RESOURCE_TYPE DM_RES (* Device Management Resource Type *)
  (* Standard: 61499-2 *)
  (* Version 0.0, 2000-05-27, JHC, Rockwell Automation *)
  VAR_INPUT
    ID : WSTRING;
  END_VAR
  FBS
    START : E_RESTART;
    MGR_FF : E_SR;
    KERNEL : DM_KRNL;
  END_FBS
  EVENT_CONNECTIONS
    START.COLD TO MGR_FF.S;
    START.WARM TO MGR_FF.S;
    START.STOP TO MGR_FF.R;
    MGR_FF.EO TO KERNEL.INIT;
  END_CONNECTIONS
  DATA_CONNECTIONS
    MGR_FF.Q TO KERNEL.QI;
    ID TO KERNEL.ID;
  END_CONNECTIONS
END_RESOURCE_TYPE
